TYPE ST_HMI_Monitor_Connections :
STRUCT
	b_ExtControllerEnabled		: BOOL;
	e_ExtConnectionState		: eConnectionState;
	s_OutputJson				: STRING(2000);
	b_IoTEnabled				: BOOL;
	e_IoTConnectionState		: eConnectionState;
	b_PsbOK						: BOOL;			
	e_ActiveController			: eControlSources;
	e_ProfinetState				: eNetcomState;
	e_EthercatState				: eNetcomState;
	r_CPUload					: REAL;
	
END_STRUCT
END_TYPE

(* stored: Version 1.1.0.1, ProductVersion 3.1.4026.18
   DUT ST_HMI_Monitor_Connections: Id {22d21adc-b3fa-4fec-9e31-c0c4b9345a6d} *)
